{attribute 'linkalways'} 
{attribute 'no_explicit_call' := 'This FB is a CLASS and must be accessed using methods or properties'}
{attribute 'enable_dynamic_creation'}
FUNCTION_BLOCK _ETcVnBarcodeSearchDirection EXTENDS EnumDatatypeBase
VAR
	localData : ETcVnBarcodeSearchDirection;
	activeData : REFERENCE TO ETcVnBarcodeSearchDirection;
	enumBaseDatatype : _UDINT(localData);
END_VAR

METHOD PRIVATE AddLocalEnumeration
VAR_INPUT
	Enumeration : T_MAXSTRING;
	Value : ETcVnBarcodeSearchDirection;
END_VAR
AddEnumeration(Enumeration, Value);
END_METHOD

PROPERTY PUBLIC Address : PVOID
GET
Address := ADR(activeData);
END_GET
END_PROPERTY

METHOD PUBLIC ClearReference
VAR_INPUT
END_VAR
activeData REF= localData;
SetBaseDatatypeReference();
END_METHOD

METHOD PUBLIC Clone : I_Datatype
VAR
    pClone : POINTER TO _ETcVnBarcodeSearchDirection;
END_VAR
pClone := __NEW(_ETcVnBarcodeSearchDirection(InitialValue := Value));
Clone := pClone^;
END_METHOD

METHOD FB_init : BOOL
VAR_INPUT
	bInitRetains : BOOL; // if TRUE, the retain variables are initialized (warm start / cold start)
	bInCopyCode : BOOL;  // if TRUE, the instance afterwards gets moved into the copy code (online change)
	InitialValue : ETcVnBarcodeSearchDirection;
END_VAR
localData := InitialValue;
AddBaseDatatype(enumBaseDatatype);
ClearReference();

AddLocalEnumeration('TCVN_BSD_ANY', ETcVnBarcodeSearchDirection.TCVN_BSD_ANY);
AddLocalEnumeration('TCVN_BSD_HORIZONTAL', ETcVnBarcodeSearchDirection.TCVN_BSD_HORIZONTAL);
AddLocalEnumeration('TCVN_BSD_VERTICAL', ETcVnBarcodeSearchDirection.TCVN_BSD_VERTICAL);
END_METHOD

PROPERTY PUBLIC Identifier : T_MAXSTRING
GET
Identifier := 'ETcVnBarcodeSearchDirection';
END_GET
END_PROPERTY

METHOD IsEnumeratorValueEqual : BOOL
VAR_INPUT
	Enumerator : I_KeyValueForwardEnumerator;
END_VAR
VAR
	storedValue : ETcVnBarcodeSearchDirection;
END_VAR
IF NOT Enumerator.TryGet(storedValue) THEN
	RETURN;
END_IF

IsEnumeratorValueEqual := storedValue = activeData;
END_METHOD

METHOD PUBLIC MakeReferenceTo
VAR_INPUT
	ReferenceTarget : REFERENCE TO ETcVnBarcodeSearchDirection;
END_VAR
activeData REF= ReferenceTarget;
SetBaseDatatypeReference();
END_METHOD

METHOD PROTECTED SetBaseDatatypeReference
VAR_INPUT
END_VAR
enumBaseDatatype.MakeReferenceTo(activeData);
END_METHOD

PROPERTY PUBLIC Size : UDINT
GET
Size := SIZEOF(activeData);
END_GET
END_PROPERTY

METHOD TryMakeReferenceTo : BOOL
VAR_INPUT
	Target : I_Datatype;
END_VAR
VAR
	targetAsEnum : I_EnumDatatype;
	pTargetData : POINTER TO ETcVnBarcodeSearchDirection;
END_VAR
IF NOT Target.TryResolveAsEnumDatatype(targetAsEnum) THEN
	RETURN;
END_IF

IF targetAsEnum.Identifier <> Identifier THEN
	RETURN;
END_IF

pTargetData := Target.Address;
activeData REF= pTargetData^;
SetBaseDatatypeReference();
TryMakeReferenceTo := TRUE;
END_METHOD

PROPERTY PUBLIC Value : ETcVnBarcodeSearchDirection
GET
Value := activeData;
END_GET
SET
activeData := Value;
END_SET
END_PROPERTY

END_FUNCTION_BLOCK

(* stored: Version 1.1.0.1, ProductVersion 3.1.4024.12
   POU _ETcVnBarcodeSearchDirection: Id {5841b578-f4eb-0af8-2e6e-61709b73c786}, SpecialFunc None
   Folder Constructor: Id {453f3c09-990d-0cd0-1476-31dfb6b9c150}
   Folder Private: Id {d29a83b9-d019-0406-3528-6cd0c31e076d}
   Folder Protected: Id {90871f83-771e-097f-2338-4962e0e94242}
   Method AddLocalEnumeration: Id {253fdc3e-5903-0310-2f9d-11049ed2e543}
   Property Address: Id {1db58ab2-38e5-0da7-01ff-41820ddd51f7}
   Get Get: Id {53833ae1-66c7-0456-181a-ce85673905ff}
   Method ClearReference: Id {af3a6bc8-b6ea-0b5d-27c1-5cf376831d06}
   Method Clone: Id {429858c4-fc2c-0464-28cf-e671907b2de4}
   Method FB_init: Id {00f45d1d-06c1-0aad-26dc-5aff5f624d5d}
   Property Identifier: Id {3859799f-0d1e-08e8-1fe3-291eee0a104a}
   Get Get: Id {c07e5eb3-f376-0473-2504-928fdae60999}
   Method IsEnumeratorValueEqual: Id {56348206-b32e-046f-3a72-2cfe9b1fcd09}
   Method MakeReferenceTo: Id {458aaac7-03fd-0b58-3c67-4319bccad0d4}
   Method SetBaseDatatypeReference: Id {efe5c9eb-e847-0d34-0ce5-638367bec757}
   Property Size: Id {a13c44c9-11f3-0f5a-3e3b-08e8f4a7726e}
   Get Get: Id {718f172a-8d47-0817-37fd-a3a2595ee83b}
   Method TryMakeReferenceTo: Id {0cdcb90c-ea18-0381-1e03-6c8fdf33b774}
   Property Value: Id {08735e48-2a69-0113-02d0-48d2f13f0b53}
   Get Get: Id {bd57febd-7e6d-0b83-309f-29f418993298}
   Set Set: Id {169343ae-86ea-09d3-11cf-570c4b214a97} *)
